// TIA Portal project "LiveTwin_Pump" (V17)

(* hardware
DEVICE "S7-1200 station_1"  S7-1200 Station
   slot 0: "Rack_0"  S7-1200 Rack  Rack  V1.0
   slot 1: "PLC_1"  CPU 1212C DC/DC/DC  6ES7 212-1AE40-0XB0  V4.4
*)

// ===== PLC "PLC_1"  CPU 1212C DC/DC/DC =====

VAR_GLOBAL   // PLC tag table "Default tag table"
   "D1" AT %I0.0 : Bool;
   "D2" AT %I0.1 : Bool;
   "A1" AT %IW64 : Int;
   "A2" AT %IW66 : Int;
   "D3" AT %I0.2 : Bool;
   "D4" AT %I0.3 : Bool;
   "D5" AT %I0.4 : Bool;
   "D6" AT %I0.5 : Bool;
   "D7" AT %I0.6 : Bool;
   "D8" AT %I0.7 : Bool;
   "Manipulator" AT %MW0 : Int;
END_VAR

VAR_GLOBAL CONSTANT   // PLC tag table "Default tag table"
   "STATE_FILL_TANK" : Int := 1;
   "STATE_HEAT_TANK" : Int := 2;
   "STATE_FILL_BOTTLE" : Int := 3;
   "STATE_SHIFT_BOTTLE" : Int := 4;
   "STATE_STOP" : Int := 5;
   "STATE_RESET" : Int := 6;
   "STATE_ERROR" : Int := 7;
END_VAR

TYPE "typeHmi"
   STRUCT
      HMI_Start : Bool;   // trigger from hmi to start
      HMI_Stop : Bool;   // trigger from hmi to stop
      HMI_Reset : Bool;   // trigger from hmi to reset
      HMI_NextBottle : Bool;   // trigger from hmi to shift bottle
      HMI_Error : Bool;   // trigger from hmi to generate error
   END_STRUCT;
END_TYPE

TYPE "typeApp"
   STRUCT
      APP_Start : Bool;   // trigger from app to start
      APP_Stop : Bool;   // trigger from app to stop
      APP_Reset : Bool;   // trigger from app to reset
      APP_QRCode : String;   // string from app containing QR code (scanning app)
   END_STRUCT;
END_TYPE

TYPE "typeSignals"
   STRUCT
      tankSignals : Struct
         actLevel : Real;   // actual level of tank [l]
         maxLevel : Bool;   // max level of tank reached
         actPressure : Real;   // actual pressure of tank [hPa]
         actTemperature : Real;   // actual temperature of tank [°C]
         maxTemperature : Bool;   // max level of temperature reached
      END_STRUCT;
      bottleSignals : Struct
         actLevel : Real;   // actual level of current bottle [l]
         maxLevel : Bool;   // max level of bottle reached
         outputTank : Real;   // Vout of Tank / Vin of bottle [m³/s]
      END_STRUCT;
      energySignals : Struct
         energyConsumptionFillingTank : Real;   // energy consumption during filling tank [Wh]
         waterConsumptionFillingTank : Real;   // water consumption during filling tank [l]
         energyConsumptionHeatingTank : Real;   // energy consumption during heating tank [Wh]
         energyConsumptionFillingBottles : Real;   // energy consumption during filling bottles [Wh]
      END_STRUCT;
      alarm : Word;   // alarm bit
   END_STRUCT;
END_TYPE

TYPE "typeOperate"
   STRUCT
      extModeActive : Bool := false;   // true = activate external model / simulation
      state : "typeState";   // operating state
      machineState : Int := 0;   // see user constants (1 = filling tank, 2 = heating tank, 3 = filling bottle, 4 = shifting bottle, 5 = stop, 6 = reset)
   END_STRUCT;
END_TYPE

TYPE "typeModel"
   STRUCT
      cycleTime : Real;   // cycle time[s]
      tank : Struct   // model struct of tank
         AT : Real;   // surface area of tank [m²]
         H : Real;   // high of tank [m]
         Vin : Real;   // incoming volume flow [l/min]
         maxLevel : Real;   // max level of tank [m³]
         roomTemperature : Real;   // room temperature of tank [°C]
         maxTemperature : Real;   // max temperature of tank [°C]
         density : Real;   // liquid density [kg/m³]
      END_STRUCT;
      bottle : Struct   // model struct of bottle
         maxLevel : Real;   // max level of bottle [m³]
         AB : Real;   // surface area of filling hole to fill bottle [m²]
      END_STRUCT;
   END_STRUCT;
END_TYPE

TYPE "typeProcess"
   STRUCT
      productId : UDInt;   // product id of current bottle
      numberProduced : UDInt;   // number of filled bottles
      numberFaulty : UDInt;   // number of faulty bottles
   END_STRUCT;
END_TYPE

TYPE "typeState"
   STRUCT
      FillingTank : Bool;   // filling tank
      HeatingTank : Bool;   // heating tank
      FillingBottle : Bool;   // filling bottle
      ShiftingBottle : Bool;   // shifting bottle
      Stop : Bool;   // stop filling
      Reset : Bool;   // reset application
      Error : Bool;   // failure
   END_STRUCT;
END_TYPE

DATA_BLOCK "LiveTwin_Pump_DB"   // DB61
{ S7_Optimized_Access := 'TRUE' }
VERSION : 0.1
// stored: InstanceOfName LiveTwin_Pump
"LiveTwin_Pump"
BEGIN
END_DATA_BLOCK

DATA_BLOCK "GlobalDB_LiveTwin"   // DB62
{ S7_Optimized_Access := 'TRUE' }
VERSION : 0.1
   VAR
      pump_speed : Real;
      flow_rate_l_min : Real;
   END_VAR
BEGIN
END_DATA_BLOCK

FUNCTION_BLOCK "LiveTwin_Pump"   // FB60, SCL
{ S7_Optimized_Access := 'TRUE' }
VERSION : 0.1
   VAR
      IEC_Timer_0_Instance : TON_TIME;
      "counter" : DInt;
      pump_speed : Real := 2500.0;
      state : USInt;
   END_VAR
   VAR_TEMP
      timer_out : Bool;
      timer_val : Time;
      timer_preset : Time;
      temp_random : Real;
   END_VAR
   VAR CONSTANT
      timer_in : Bool := true;
   END_VAR
BEGIN
   #IEC_Timer_0_Instance(IN := #timer_in,
                         PT := T#10ms,
                         Q => #timer_out,
                         ET => #timer_val);

   IF #timer_out THEN
       #counter := #counter + 1;
       RESET_TIMER(#IEC_Timer_0_Instance);
   END_IF;

   IF #counter >= 500 THEN
       #counter := 0;
       IF #state <= 2 THEN
           #state := #state + 1;
       ELSE
           #state := 0;
       END_IF;
   END_IF;

   "Random_Number"(Min := -1,
                   Max := 1,
                   RandomNumber => #temp_random);

   CASE #state OF
       0:
           #pump_speed := #pump_speed + 0.2;
       1:
           #pump_speed := #pump_speed + #temp_random * 0.2;
       2:
           IF #pump_speed >= 2510 THEN
               #pump_speed := #pump_speed - 0.21;
           END_IF;
       3:
           #pump_speed := #pump_speed + #temp_random * 0.2;
           IF #pump_speed < 2500 THEN
               #pump_speed := 2500;
           END_IF;
   END_CASE;

   "GlobalDB_LiveTwin".pump_speed := #pump_speed;
END_FUNCTION_BLOCK

FUNCTION "Random_Number" : Void   // FC3, SCL
{ S7_Optimized_Access := 'TRUE' }
VERSION : 0.1
   VAR_INPUT
      Min : Int;
      Max : Int;
   END_VAR
   VAR_OUTPUT
      RandomNumber : Int;
   END_VAR
   VAR_TEMP
      range : Int;
      tmp : Int;
      rdsys : DTL;
      ret : Int;
   END_VAR
BEGIN
   // generate random number
   #ret := RD_SYS_T(#rdsys);
   #tmp := UDINT_TO_INT(#rdsys.NANOSECOND);
   IF #tmp < 0 THEN
       #tmp := #tmp * - 1;
   END_IF;

   "Manipulator" := "Manipulator" + 1;

   IF "Manipulator" = 10 THEN
       "Manipulator" := 1;
   END_IF;

   #tmp := #tmp / "Manipulator";

   #range := #Max - #Min;

   #tmp := #tmp MOD (#range + 1);
   #RandomNumber := #tmp + #Min;
END_FUNCTION

ORGANIZATION_BLOCK "Main"   // OB1, LAD, ProgramCycle
TITLE = "Main Program Sweep (Cycle)"
{ S7_Optimized_Access := 'TRUE' }
VERSION : 0.1
   VAR_INPUT
      Initial_Call : Bool;   // Initial call of this OB
      Remanence : Bool;   // =True, if remanent data are available
   END_VAR
BEGIN

REGION Network 1
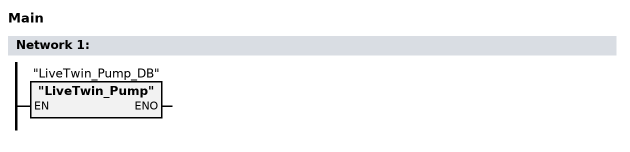
   RUNG wire#powerrail
      "LiveTwin_Pump_DB"()
   END_RUNG
   // the same network as SCL:
   "LiveTwin_Pump_DB"();   // "LiveTwin_Pump"
END_REGION
END_ORGANIZATION_BLOCK